% RSLogix 500 project SEND_BITS_BAK013.RSS, saved by version 8.10.00.18 %
PROJECT "UNTITLED"    % processor: Bul.1763 MicroLogix 1100 Series B %

PROGRAM FILES
  LAD 2   3 rungs

DATA FILES
  O0 OUTPUT  4 elements
  I1 INPUT  6 elements
  S2 STATUS  66 elements
  B3 BINARY  1 elements
  T4 TIMER  1 elements
  C5 COUNTER  1 elements
  R6 CONTROL  2 elements
  N7 INTEGER  4 elements
  F8 FLOAT  1 elements

LADDER 2
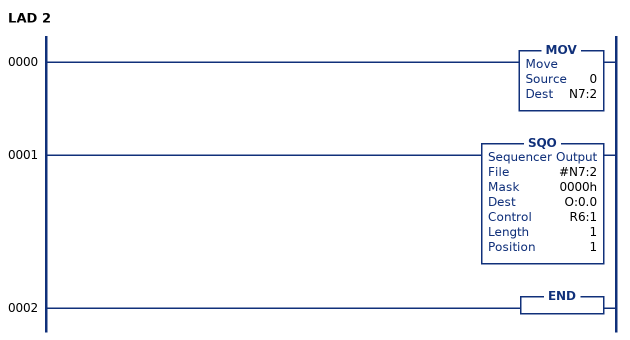
% Rung: 0 %
SOR MOV 0 N7:2 EOR
% Rung: 1 %
SOR SQO #N7:2 0000h O:0.0 R6:1 1 1 EOR
% Rung: 2 %
SOR END EOR

DATA TABLE (non-zero values as saved)
DATA R6
% .LEN .POS %
% R6:1 % 1 1
